(* PLC project Automatic_ScrewDriver_Line.project, CODESYS CODESYS V3.5 SP21 Patch 5 *)
(* stored: creationDateTime 2026-09-30T17:02:56.3790076, modificationDateTime 2026-09-30T17:02:44.4882995 *)

{attribute 'qualified_only'}
{attribute 'strict'}
TYPE JobState : (Idle := 1, Reset, ReadingTargetPosition, MovingToTargetPosition, MovingToBase, MovingZaxisToTool, ProcessingTool, MovingZaxisToBase, Error);
END_TYPE

TYPE Screw : STRUCT
  PositionMm : REAL;  (* in mm *)
  AngleDeg : DINT;  (* in ° *)
END_STRUCT;
END_TYPE

{attribute 'qualified_only'}
{attribute 'strict'}
TYPE ErrorCode : (NoError := 0, EnablementError, ScrewNotReleased, TargetNotReached, SpindleError, CobotNotConnected, CobotMovementNotReached, RtcNotAvailable);
END_TYPE

{attribute 'qualified_only'}
{attribute 'strict'}
TYPE ActionResult : (Busy := 1, Done, Failed);
END_TYPE

{attribute 'qualified_only'}
{attribute 'strict'}
TYPE MoverState : (Idle := 0, WaitingEcho, Moving, WaitingDoneReleased);
END_TYPE

TYPE JobReport : STRUCT
  JobId : UDINT;
  StartedAt : DT;
  FinishedAt : DT;
  ScrewsOk : INT;
  ScrewsFailed : INT;
  FailedScrews : ScrewList;
  Completed : BOOL;  (* TRUE = all screws processed, FALSE = aborted by operator *)
END_STRUCT;
END_TYPE

TYPE ScrewList : ARRAY[1..5] OF Screw;
END_TYPE

INTERFACE I_Actuator
METHOD Enable : BOOL
END_METHOD
METHOD Disable : BOOL
END_METHOD
END_INTERFACE

INTERFACE I_Mover
METHOD MoveToPosition : BOOL
  VAR_INPUT
    Position : REAL;
  END_VAR
END_METHOD
END_INTERFACE

INTERFACE I_Tool
METHOD ProcessTool : BOOL
  VAR_INPUT
    Angle : DINT;
  END_VAR
END_METHOD
END_INTERFACE

INTERFACE I_Resettable
METHOD Reset : BOOL
END_METHOD
END_INTERFACE

INTERFACE I_Diagnosable
METHOD GetError : ErrorCode
END_METHOD
METHOD ClearError : BOOL
END_METHOD
END_INTERFACE

INTERFACE I_ReportSink
METHOD PublishReport : BOOL
  VAR_INPUT
    Report : JobReport;
  END_VAR
END_METHOD
END_INTERFACE

INTERFACE I_Device
END_INTERFACE

PROGRAM PLC_PRG
  VAR
    _InitDone : BOOL;
    _JobManager : FB_JobManager;
    _UserInterface : FB_UserInterface;
    _JobSelector : FB_JobSelector;
    _Conveyor : FB_ConveyorElectrical;
    _Cobot : FB_Cobot;
    _zAxis : FB_zAxis;
    _Spindle : FB_Spindle;
    _ReportJob : FB_ReportJob;
    _LogSink : FB_LogSink;
  END_VAR

                    IF NOT _InitDone THEN
	_InitDone := InitPous();
END_IF


_JobManager.RunJob();


//I/O's connection: Machine -> Material
//For Conveyor:
IO_Simulation.MoverEnable := _Conveyor.MoverEnable;
IO_Simulation.MoverExecuteFor :=  _Conveyor.MoverExecuteFor;
IO_Simulation.MoverExecuteBac :=  _Conveyor.MoverExecuteBac;
// For Robot:
IO_Cobot.Cmd_TargetPos01mm := INT_TO_WORD(_Cobot.MoverTarget);   // 0..5000: no sign issue
IO_Cobot.Cmd_Start := _Cobot.MoverExecute;
IO_Cobot.Cmd_Enable := _Cobot.MoverEnable;
// For Z valve
IO_Simulation.zValve := _zAxis.zValve;
// For Spindle
IO_Simulation.SpindleEnable := _Spindle.SpindleEnable;
IO_Simulation.SpindleExecute := _Spindle.SpindleExecute;
IO_Simulation.SpindleExecuteTime := _Spindle.SpindleExecuteTime;

// Simulation
PRG_PlantSim();

//I/O's connection: Material -> Machine
//For Conveyor:
_Conveyor.MoverActPos := IO_Simulation.MoverActPos;
_Conveyor.MoverReady := IO_Simulation.MoverReady; 
// For cobot:
_Cobot.MoverPosEcho := WORD_TO_INT(IO_Cobot.Sts_TargetPosEcho01mm);
_Cobot.MoverDone := IO_Cobot.Sts_Done;
_Cobot.MoverHeartbeat := WORD_TO_INT(IO_Cobot.Sts_Heartbeat);
// For Z valve
_zAxis.ScrewEngaged := IO_Simulation.ScrewEngaged;
_zAxis.ScrewReleased := IO_Simulation.ScrewReleased;
_zAxis.zDown := IO_Simulation.zDown;
// For Spindle
_Spindle.SpindleReady := IO_Simulation.SpindleReady;
_Spindle.SpindleDone := IO_Simulation.SpindleDone;




                  

METHOD InitPous : BOOL
  VAR
    _Mover : I_Mover;
  END_VAR
                          // Injection of dependencies
IF Machine_Constants.USE_COBOT THEN
	_Mover := _Cobot;
ELSE
	_Mover := _Conveyor;
END_IF

_ReportJob.AddSink(_LogSink);

InitPous := _JobManager.Init(
	UserInterface := _UserInterface,
	JobSelector := _JobSelector,
	Mover:= _Mover,
	zAxis := _zAxis,
	Spindle := _Spindle,
	ReportJob := _ReportJob);
                        
END_METHOD
END_PROGRAM

FUNCTION_BLOCK FB_FunctionBlock_Base IMPLEMENTS I_Resettable, I_Diagnosable
  VAR
    _Error : ErrorCode;
  END_VAR

                    
                  

{attribute 'abstract'}
METHOD Reset : BOOL
                          
                        
END_METHOD

METHOD RaiseError : BOOL
  VAR_INPUT
    Error : ErrorCode;
  END_VAR
                          RaiseError := FALSE;

IF _Error = ErrorCode.NoError THEN
	_Error := Error;
	Trace(CmpLog.LogClass.LOG_ERROR, ErrorCodeToString(Error));
	RaiseError := TRUE;
END_IF

                        
END_METHOD

METHOD GetError : ErrorCode
                          GetError := _Error;
                        
END_METHOD

METHOD ClearError : BOOL
                          _Error := ErrorCode.NoError;
ClearError := TRUE;
                        
END_METHOD

METHOD HasError : BOOL
                          HasError := (_Error <> ErrorCode.NoError);
                        
END_METHOD
END_FUNCTION_BLOCK

FUNCTION_BLOCK FB_JobManager EXTENDS FB_FunctionBlock_Base
  VAR
    _InitDone : BOOL;
    _state : JobState;
    _ActiveError : ErrorCode;
    _Stop : BOOL;
    _Reseters : ARRAY[1..6] OF I_Resettable;
    _Diagnosable : ARRAY[1..6] OF I_Diagnosable;
    _i : DINT;
    _UserInterface : REFERENCE TO FB_UserInterface;
    _JobSelector : REFERENCE TO FB_JobSelector;
    _Mover : I_Mover;
    _zAxis : REFERENCE TO FB_zAxis;
    _Spindle : REFERENCE TO FB_Spindle;
    _ReportJob : REFERENCE TO FB_ReportJob;
    _SpindleOk : BOOL;
    _MoverOk : BOOL;
  END_VAR

                    
                  

METHOD Reset : BOOL
                          ClearError();
Reset := TRUE;

                        
END_METHOD

METHOD Init : BOOL
  VAR_INPUT
    UserInterface : REFERENCE TO FB_UserInterface;
    JobSelector : REFERENCE TO FB_JobSelector;
    Mover : I_Mover;
    zAxis : REFERENCE TO FB_zAxis;
    Spindle : REFERENCE TO FB_Spindle;
    ReportJob : REFERENCE TO FB_ReportJob;
  END_VAR
                          _UserInterface REF= UserInterface;
_JobSelector REF= JobSelector;
_Mover := Mover;
_zAxis REF= zAxis;
_Spindle REF= Spindle;
_ReportJob REF= ReportJob;

// Reseters
_Reseters[1] := _UserInterface;
_Reseters[2] := _JobSelector;
_Reseters[3] := _Mover;
_Reseters[4] := _zAxis;
_Reseters[5] := _Spindle;
_Reseters[6] := _ReportJob;

// Diagnosable
_Diagnosable[1] := _UserInterface;
_Diagnosable[2] := _JobSelector;
_Diagnosable[3] := _Mover;
_Diagnosable[4] := _zAxis;
_Diagnosable[5] := _Spindle;
_Diagnosable[6] := _ReportJob;

_InitDone := TRUE;
Init := TRUE;
                        
END_METHOD

METHOD DisableAll : BOOL
                          _SpindleOk := _Spindle.Disable();
_MoverOk   := _Mover.Disable();
DisableAll := _SpindleOk AND _MoverOk;
                        
END_METHOD

METHOD EnableAll : BOOL
                          _SpindleOk := _Spindle.Enable();
_MoverOk   := _Mover.Enable();
EnableAll  := _SpindleOk AND _MoverOk;

                        
END_METHOD

METHOD ResetAll : BOOL
                          ResetAll := TRUE;

FOR _i := 1 TO UPPER_BOUND(_Reseters, 1) DO
    IF NOT _Reseters[_i].Reset() THEN
        ResetAll := FALSE;
    END_IF
END_FOR
                        
END_METHOD

METHOD CheckErrors : ErrorCode
                          CheckErrors := ErrorCode.NoError;

FOR _i := 1 TO UPPER_BOUND(_Diagnosable, 1) DO
    IF _Diagnosable[_i].GetError() <> ErrorCode.NoError
       AND CheckErrors = ErrorCode.NoError THEN
        CheckErrors := _Diagnosable[_i].GetError();
    END_IF
END_FOR
                        
END_METHOD

METHOD RunJob : BOOL
                          IF NOT _InitDone THEN
	RETURN;
END_IF

_ActiveError := CheckErrors();
_Stop := _UserInterface.IsStopRequired();
		  
IF _ActiveError <> ErrorCode.NoError AND _state <> JobState.Reset THEN
    _state := JobState.Error;
END_IF

IF _state <> JobState.Reset AND _state <> JobState.Error THEN
    EnableAll();
ELSE
    DisableAll();
END_IF

CASE _state OF
	JobState.Reset :
		IF ResetAll() THEN
			_state := JobState.Idle;
		END_IF
	JobState.Idle:
		IF _Stop THEN
			_state := JobState.Reset;
		ELSIF _zAxis.Retract() THEN
        	IF _UserInterface.IsStartRequired() THEN
            _ReportJob.Reset();
			_ReportJob.JobStart();
            _state := JobState.ReadingTargetPosition;
        	END_IF
    	END_IF
	JobState.ReadingTargetPosition :
		IF _JobSelector.ReturnScrew() THEN
			_state:= JobState.MovingToTargetPosition;
		ELSE
			_state := JobState.MovingToBase;
		END_IF
	JobState.MovingToTargetPosition :
		IF _Mover.MoveToPosition(_JobSelector.CurrentScrew.PositionMm) THEN
			_state:= JobState.MovingZaxisToTool;
		END_IF
	JobState.MovingZaxisToTool :
		    CASE _zAxis.Engage() OF
        		ActionResult.Done:
            		_state := JobState.ProcessingTool;
				ActionResult.Failed:
            		_ReportJob.FailScrew(_JobSelector.CurrentScrew);
					_state := JobState.MovingZaxisToBase;
    		END_CASE
	JobState.ProcessingTool :
		IF _Spindle.ProcessTool(_JobSelector.CurrentScrew.AngleDeg) THEN		
			_ReportJob.SuccessScrew(_JobSelector.CurrentScrew);
			_state:= JobState.MovingZaxisToBase;
		END_IF
	JobState.MovingZaxisToBase :
		IF _zAxis.Retract() THEN
			_state:= JobState.ReadingTargetPosition;
		END_IF
	JobState.MovingToBase :
		IF _Mover.MoveToPosition(0)  THEN
			_state := JobState.Idle;
			_ReportJob.JobEnd();
		END_IF
	JobState.Error :
		IF _Stop THEN
			_state := JobState.Reset;
		END_IF
END_CASE

// Stop during a job = abort: publish the partial report, then reset every component.
// The next Start begins a fresh job from the first screw.
IF _Stop
   AND _state <> JobState.Idle
   AND _state <> JobState.Reset
   AND _state <> JobState.Error THEN
	_ReportJob.JobAborted();
	_state := JobState.Reset;
END_IF

                        
END_METHOD
END_FUNCTION_BLOCK

FUNCTION_BLOCK FB_UserInterface EXTENDS FB_FunctionBlock_Base
  VAR_INPUT
    StartRequest : BOOL;
    StopRequest : BOOL;
  END_VAR
  VAR
    _Start_Trig : R_TRIG;
    _Stop_Trig : R_TRIG;
  END_VAR

                    
                  

METHOD Reset : BOOL
                          ClearError();
Reset := TRUE;
                        
END_METHOD

METHOD IsStartRequired : BOOL
                          _Start_Trig(CLK := StartRequest);
IsStartRequired := _Start_Trig.Q;

                        
END_METHOD

METHOD IsStopRequired : BOOL
                          _Stop_Trig(CLK := StopRequest);
IsStopRequired := _Stop_Trig.Q;
                        
END_METHOD
END_FUNCTION_BLOCK

FUNCTION_BLOCK FB_JobSelector EXTENDS FB_FunctionBlock_Base
  VAR_INPUT
    ArrScrews : ScrewList := [(PositionMm := 100.0, AngleDeg := 90), (PositionMm := 130.0, AngleDeg := 600), (PositionMm := 185.0, AngleDeg := -180), (PositionMm := 27.0, AngleDeg := 360), (PositionMm := 300.0, AngleDeg := 720)];
  END_VAR
  VAR_OUTPUT
    CurrentScrew : Screw;
    Job_Done : BOOL;
  END_VAR
  VAR
    _TableIndex : INT := 0;
  END_VAR

                    
                  

METHOD Reset : BOOL
                          ClearError();
_TableIndex := 0;
Job_Done := FALSE;

Reset := TRUE;
                        
END_METHOD

METHOD ReturnScrew : BOOL
                          ReturnScrew := FALSE;


IF SelectNextScrew() THEN
	CurrentScrew := ArrScrews[_TableIndex];
	ReturnScrew := TRUE;
ELSE
	CurrentScrew.PositionMm := 0.0;
	CurrentScrew.AngleDeg := 0;
END_IF

                        
END_METHOD

METHOD SelectNextScrew : BOOL
                          // Method responsible for incrementing _TableIndex
SelectNextScrew := FALSE;
Job_Done := FALSE;
IF _TableIndex < UPPER_BOUND(ArrScrews, 1) THEN
	_TableIndex := _TableIndex + 1;
	SelectNextScrew := TRUE;
ELSE
	_TableIndex := 0;
	Job_Done := TRUE;
END_IF
                        
END_METHOD
END_FUNCTION_BLOCK

FUNCTION_BLOCK FB_ConveyorElectrical EXTENDS FB_FunctionBlock_Base IMPLEMENTS I_Mover
  VAR_INPUT
    MoverActPos : REAL;
    MoverReady : BOOL;
  END_VAR
  VAR_OUTPUT
    MoverEnable : BOOL;
    MoverExecuteFor : BOOL;
    MoverExecuteBac : BOOL;
  END_VAR
  VAR
    _MoverTarget : REAL;
    _TimerEnablement : TON;
    _TimerMoveLinear : TON;
  END_VAR

                    
                  

METHOD Reset : BOOL
                          ClearError();
Disable();
MoverExecuteFor := FALSE;
MoverExecuteBac := FALSE;
_MoverTarget :=  0.0;
_TimerEnablement(IN := FALSE, PT := T#1S);
_TimerMoveLinear(IN := FALSE, PT := T#100S);
Reset := TRUE;
                        
END_METHOD

METHOD MoveToPosition : BOOL
  VAR_INPUT
    Position : REAL;
  END_VAR
                          MoveToPosition := FALSE;

_MoverTarget := Position;


IF _TimerMoveLinear.Q THEN
	RaiseError(ErrorCode.TargetNotReached);
ELSIF _MoverTarget - MoverActPos >= 1 THEN
	MoverExecuteFor := TRUE;
ELSIF _MoverTarget - MoverActPos <= -1 THEN
	MoverExecuteBac := TRUE;
ELSE
	MoveToPosition := TRUE;
	MoverExecuteFor := FALSE;
	MoverExecuteBac := FALSE;
END_IF

_TimerMoveLinear(IN := (MoverExecuteFor OR MoverExecuteBac), PT := T#100S);

                        
END_METHOD

METHOD Enable : BOOL
                          Enable := FALSE;

MoverEnable := TRUE;
_TimerEnablement(IN := MoverEnable AND NOT MoverReady, PT := T#1S);

IF MoverReady THEN
	Enable := TRUE;
ELSIF _TimerEnablement.Q THEN
	RaiseError(ErrorCode.EnablementError);
END_IF

                        
END_METHOD

METHOD Disable : BOOL
                          MoverEnable := FALSE;
Disable := TRUE;
                        
END_METHOD
END_FUNCTION_BLOCK

FUNCTION_BLOCK FB_zAxis EXTENDS FB_FunctionBlock_Base
  VAR_INPUT
    zDown : BOOL;
    ScrewEngaged : BOOL;
    ScrewReleased : BOOL;
  END_VAR
  VAR_OUTPUT
    zValve : BOOL;
  END_VAR
  VAR
    _timerUp : TON;
    _timerDown : TON;
  END_VAR

                    
                  

METHOD Reset : BOOL
                          ClearError();

zValve := FALSE;

IF zDown THEN
	Reset := TRUE;
END_IF

_timerUp(IN := FALSE, PT := T#5S);
_timerDown(IN := FALSE, PT := T#5S);
                        
END_METHOD

METHOD Engage : ActionResult
                          Engage := ActionResult.Busy;
zValve := TRUE;

_timerUp(IN := zValve AND NOT ScrewEngaged, PT := T#5S);
_timerDown(IN := FALSE, PT := T#5S);

IF ScrewEngaged THEN
	Engage := ActionResult.Done;
ELSIF _timerUp.Q THEN
	Engage := ActionResult.Failed;
END_IF


                        
END_METHOD

METHOD Retract : BOOL
                          Retract := FALSE;
zValve := FALSE;

_timerDown(IN := NOT zValve AND NOT (zDown AND ScrewReleased), PT := T#5S);
_timerUp(IN := FALSE, PT := T#5S);

IF zDown AND ScrewReleased THEN
    Retract := TRUE;
ELSIF _timerDown.Q THEN
	RaiseError(ErrorCode.ScrewNotReleased);
END_IF


                        
END_METHOD
END_FUNCTION_BLOCK

FUNCTION_BLOCK FB_Spindle EXTENDS FB_FunctionBlock_Base IMPLEMENTS I_Actuator
  VAR_INPUT
    SpeedDegPerSec : DINT := Machine_Constants.TOOL_SPEED;
    SpindleReady : BOOL;
    SpindleDone : BOOL;
  END_VAR
  VAR_OUTPUT
    SpindleEnable : BOOL;
    SpindleExecute : BOOL;
    SpindleExecuteTime : TIME;
  END_VAR
  VAR
    _AngleTarget : DINT;
    _Started : BOOL;
    _TimerEnablement : TON;
    _TimerProcessTool : TON;
  END_VAR

                    
                  

METHOD Reset : BOOL
                          ClearError();
Disable();
SpindleEnable := FALSE;
SpindleExecute := FALSE;
SpindleExecuteTime := T#0S;
_AngleTarget := 0;
_Started := FALSE;
_TimerEnablement(IN := FALSE, PT := T#1S);
_TimerProcessTool(IN := FALSE, PT := T#20S);
Reset := TRUE;
                        
END_METHOD

METHOD ProcessTool : BOOL
  VAR_INPUT
    Angle : DINT;
  END_VAR
                          ProcessTool := FALSE;
_TimerProcessTool(IN := SpindleExecute AND NOT SpindleDone, PT := T#20S);
_AngleTarget := ABS(Angle); 

IF NOT _Started AND SpindleEnable THEN
	SpindleExecuteTime := DINT_TO_TIME(_AngleTarget*1000/SpeedDegPerSec);
	SpindleExecute := TRUE;
	_Started := TRUE;
ELSIF SpindleDone THEN
	SpindleExecute := FALSE;
	_Started := FALSE;
	ProcessTool := TRUE;
ELSIF _TimerProcessTool.Q THEN
	RaiseError(ErrorCode.SpindleError);
END_IF


                        
END_METHOD

METHOD Enable : BOOL
                          Enable := FALSE;

SpindleEnable := TRUE;
_TimerEnablement(IN := SpindleEnable AND NOT SpindleReady, PT := T#1S);

IF SpindleReady THEN
	Enable := TRUE;
ELSIF _TimerEnablement.Q THEN
	RaiseError(ErrorCode.EnablementError);
END_IF
                        
END_METHOD

METHOD Disable : BOOL
                          SpindleEnable := FALSE;
Disable := TRUE;
                        
END_METHOD
END_FUNCTION_BLOCK

PROGRAM PRG_PlantSim
  VAR
    _Increment : REAL := 1;
    _ZAxisMovingTimeUp : TON;
    _ZAxisMovingTimeDown : TON;
    _SpindleMovingTime : TON;
  END_VAR

                    // Conveyor
IO_Simulation.MoverReady := IO_Simulation.MoverEnable
                                   AND NOT IO_Simulation.SimFail_MoverReady;
IF IO_Simulation.MoverExecuteFor AND IO_Simulation.MoverEnable
   AND NOT IO_Simulation.SimFail_MoverBlocked THEN
    IO_Simulation.MoverActPos := IO_Simulation.MoverActPos + _Increment;
ELSIF IO_Simulation.MoverExecuteBac AND IO_Simulation.MoverEnable
   AND NOT IO_Simulation.SimFail_MoverBlocked THEN
    IO_Simulation.MoverActPos := IO_Simulation.MoverActPos - _Increment;
END_IF

// Z Axis
_ZAxisMovingTimeUp(IN := IO_Simulation.zValve, PT := T#1S);
IO_Simulation.ScrewEngaged := _ZAxisMovingTimeUp.Q
                                     AND NOT IO_Simulation.SimFail_ScrewEngaged;
_ZAxisMovingTimeDown(IN := NOT IO_Simulation.zValve, PT := T#1S);
IO_Simulation.ScrewReleased := _ZAxisMovingTimeDown.Q
                                      AND NOT IO_Simulation.SimFail_ScrewReleased;
// zDown is not filtered: the cylinder physically retracts even if the bit stays engaged
IO_Simulation.zDown := _ZAxisMovingTimeDown.Q;

// Spindle
IO_Simulation.SpindleReady := IO_Simulation.SpindleEnable;
_SpindleMovingTime(IN := IO_Simulation.SpindleExecute
                         AND IO_Simulation.SpindleEnable,
                   PT := IO_Simulation.SpindleExecuteTime);
IO_Simulation.SpindleDone := _SpindleMovingTime.Q
                                    AND NOT IO_Simulation.SimFail_SpindleDone;
                  
END_PROGRAM

FUNCTION_BLOCK FB_ReportJob EXTENDS FB_FunctionBlock_Base
  VAR
    _NbSuccess : INT := 0;
    _NbFail : INT := 0;
    _FailedScrews : ScrewList;
    _SuccessfulScrews : ScrewList;
    _JobDone : BOOL;
    _JobId : UDINT;
    _StartedAt : DT;
    _FinishedAt : DT;
    _Sinks : ARRAY[1..3] OF I_ReportSink;
    _EmptyScrewList : ScrewList;
  END_VAR

                    
                  

METHOD Reset : BOOL
                          ClearError();
_NbSuccess := 0;
_NbFail := 0;
_JobDone := FALSE;

_FailedScrews     := _EmptyScrewList;
_SuccessfulScrews := _EmptyScrewList;

Reset := TRUE;
                        
END_METHOD

METHOD JobEnd : BOOL
                          _FinishedAt := Now();

Trace(CmpLog.LogClass.LOG_INFO, 'Job Done');

JobEnd := SendReportToSinks(Completed := TRUE);
                        
END_METHOD

METHOD SuccessScrew : BOOL
  VAR_INPUT
    SuccessfulScrew : Screw;
  END_VAR
                          SuccessScrew := FALSE;

IF _NbSuccess < UPPER_BOUND(_SuccessfulScrews, 1) THEN
	_NbSuccess := _NbSuccess + 1;
	_SuccessfulScrews[_NbSuccess] := SuccessfulScrew;
	SuccessScrew := TRUE;
END_IF

Trace(CmpLog.LogClass.LOG_INFO,
        CONCAT('Screw successfully processed at position ', REAL_TO_STRING(SuccessfulScrew.PositionMm)));
                        
END_METHOD

METHOD FailScrew : BOOL
  VAR_INPUT
    FailedScrew : Screw;
  END_VAR
                          FailScrew := FALSE;

IF _NbFail < UPPER_BOUND(_FailedScrews, 1) THEN
	_NbFail := _NbFail + 1;
	_FailedScrews[_NbFail] := FailedScrew;
	FailScrew := TRUE;
END_IF

Trace(CmpLog.LogClass.LOG_WARNING,
        CONCAT('Screw missed at position ', REAL_TO_STRING(FailedScrew.PositionMm)));
                        
END_METHOD

METHOD JobStart : BOOL
                          _JobId      := _JobId + 1;
_StartedAt  := Now();
_FinishedAt := DT#1970-01-01-00:00:00;

Trace(CmpLog.LogClass.LOG_INFO, 'Job Started');

JobStart := TRUE;
                        
END_METHOD

METHOD JobAborted : BOOL
                          _FinishedAt := Now();

Trace(CmpLog.LogClass.LOG_WARNING, 'Job Aborted');

JobAborted := SendReportToSinks(Completed := FALSE);
                        
END_METHOD

METHOD AddSink : BOOL
  VAR_INPUT
    Sink : I_ReportSink;
  END_VAR
  VAR
    _i : DINT;
  END_VAR
                          AddSink := FALSE;

FOR _i := 1 TO UPPER_BOUND(_Sinks, 1) DO
	IF _Sinks[_i] = 0 THEN
		_Sinks[_i] := Sink;
		AddSink := TRUE;
		RETURN;
	END_IF
END_FOR
                        
END_METHOD

METHOD SendReportToSinks : BOOL
  VAR_INPUT
    Completed : BOOL;  (* TRUE = job finished normally, FALSE = aborted by operator *)
  END_VAR
  VAR
    _report : JobReport;
    _i : DINT;
  END_VAR
                          _report.JobId        := _JobId;
_report.StartedAt    := _StartedAt;
_report.FinishedAt   := _FinishedAt;
_report.ScrewsOk     := _NbSuccess;
_report.ScrewsFailed := _NbFail;
_report.FailedScrews := _FailedScrews;
_report.Completed := Completed;

SendReportToSinks := TRUE;

FOR _i := 1 TO UPPER_BOUND(_Sinks, 1) DO
	IF _Sinks[_i] <> 0 THEN
		IF NOT _Sinks[_i].PublishReport(_report) THEN
			SendReportToSinks := FALSE;
		END_IF
	END_IF
END_FOR
                        
END_METHOD

METHOD Now : DT
  VAR
    _sec : UDINT;
    _res : RTS_IEC_RESULT;
  END_VAR
                          _sec := SysTimeRtcGet(_res);

IF _res = Errors.ERR_OK THEN
	Now := UDINT_TO_DT(_sec);
ELSE
	Now := DT#1970-01-01-00:00:00;
	RaiseError(ErrorCode.RtcNotAvailable);
END_IF
                        
END_METHOD
END_FUNCTION_BLOCK

FUNCTION ErrorCodeToString : STRING
  VAR_INPUT
    Code : ErrorCode;
  END_VAR

                    CASE Code OF
	ErrorCode.NoError :
		ErrorCodeToString := 'No Error';
	ErrorCode.EnablementError:
		ErrorCodeToString := 'Enablement Error';
	ErrorCode.ScrewNotReleased:
		ErrorCodeToString := 'Screw Not Released';
	ErrorCode.TargetNotReached:
		ErrorCodeToString := 'Target Not Reached';
	ErrorCode.SpindleError:
		ErrorCodeToString := 'Spindle Error';
	ErrorCode.CobotNotConnected:
		ErrorCodeToString := 'Cobot Not Connected';
	ErrorCode.CobotMovementNotReached:
		ErrorCodeToString := 'Cobot Movement Not Reached';
	ErrorCode.RtcNotAvailable:
		ErrorCodeToString := 'Rtc Not Available';
ELSE
		ErrorCodeToString := 'Unknown Error';	
END_CASE
                  
END_FUNCTION

FUNCTION_BLOCK FB_Cobot EXTENDS FB_FunctionBlock_Base IMPLEMENTS I_Mover
  VAR_INPUT
    MoverPosEcho : INT;  (* Echo to ensure synchronisation with MoverTarget *)
    MoverDone : BOOL;
    MoverHeartbeat : INT;  (* Watchdog counter to make sure Cobot connection is not lost *)
  END_VAR
  VAR_OUTPUT
    MoverEnable : BOOL;
    MoverTarget : INT;
    MoverExecute : BOOL;
  END_VAR
  VAR
    _state : MoverState := MoverState.Idle;
    _TimerEcho : TON;
    _TimerMove : TON;
    _TimerEnablement : TON;
    _LastHeartbeat : INT;
    _HbTimer : TON;
    _Alive : BOOL;
    _HbChanged : BOOL;
  END_VAR

                    
                  

METHOD Reset : BOOL
                          ClearError();
Disable();
MoverTarget :=  0;
_state := MoverState.Idle;
_TimerEnablement(IN := FALSE, PT := T#1S);
_TimerEcho(IN := FALSE, PT := T#2S);
_TimerMove(IN := FALSE, PT := T#30S);
_HbTimer(IN := FALSE, PT := T#500MS);

Reset := TRUE;
                        
END_METHOD

METHOD MoveToPosition : BOOL
  VAR_INPUT
    Position : REAL;
  END_VAR
                          MoveToPosition := FALSE;

CASE _state OF

	MoverState.Idle:
		// Never start a cycle while the robot still asserts Done from a previous one
		IF NOT MoverDone THEN
			MoverTarget  := REAL_TO_INT(Position * 10.0);
			MoverExecute := FALSE;
			_state := MoverState.WaitingEcho;
		END_IF

	MoverState.WaitingEcho:
		IF MoverPosEcho = MoverTarget THEN
			MoverExecute := TRUE;
			_state := MoverState.Moving;
		ELSIF _TimerEcho.Q THEN
			RaiseError(ErrorCode.CobotNotConnected);
		END_IF

	MoverState.Moving:
		IF MoverDone THEN
			MoverExecute := FALSE;
			_state := MoverState.WaitingDoneReleased;
		ELSIF _TimerMove.Q THEN
			RaiseError(ErrorCode.CobotMovementNotReached);
		END_IF

	MoverState.WaitingDoneReleased:
		IF NOT MoverDone THEN
			MoveToPosition := TRUE;
			_state := MoverState.Idle;
		END_IF

END_CASE

_TimerEcho(IN := (_state = MoverState.WaitingEcho), PT := T#2S);
_TimerMove(IN := (_state = MoverState.Moving), PT := T#30S);

                        
END_METHOD

METHOD Enable : BOOL
                          _HbChanged := (MoverHeartbeat <> _LastHeartbeat);
_LastHeartbeat := MoverHeartbeat;
_HbTimer(IN := NOT _HbChanged, PT := T#500MS);
_Alive := NOT _HbTimer.Q;

Enable := FALSE;
MoverEnable := TRUE;

_TimerEnablement(IN := NOT _Alive, PT := T#1S);

IF _Alive THEN
	Enable := TRUE;
ELSIF _TimerEnablement.Q THEN
	RaiseError(ErrorCode.CobotNotConnected);
END_IF

                        
END_METHOD

METHOD Disable : BOOL
                          MoverEnable  := FALSE;
MoverExecute := FALSE;
Disable := TRUE;
                        
END_METHOD
END_FUNCTION_BLOCK

FUNCTION_BLOCK FB_LogSink IMPLEMENTS I_ReportSink

                    
                  

METHOD PublishReport : BOOL
  VAR_INPUT
    Report : JobReport;
  END_VAR
  VAR
    _msg : STRING(255);
  END_VAR
                          _msg := CONCAT('Job ', UDINT_TO_STRING(Report.JobId));
_msg := CONCAT(_msg,   ' finished: ');
_msg := CONCAT(_msg,   INT_TO_STRING(Report.ScrewsOk));
_msg := CONCAT(_msg,   ' ok, ');
_msg := CONCAT(_msg,   INT_TO_STRING(Report.ScrewsFailed));
_msg := CONCAT(_msg,   ' failed');

Trace(CmpLog.LogClass.LOG_INFO, _msg);

PublishReport := TRUE;
                        
END_METHOD
END_FUNCTION_BLOCK

FUNCTION Trace : BOOL
  VAR_INPUT
    Severity : UDINT;  (* LogClass.LOG_INFO / LOG_WARNING / LOG_ERROR *)
    Msg : STRING(255);
  END_VAR

                    LogAdd(
	hLogger   := CmpLog.LogConstants.LOG_STD_LOGGER,
	stCmpName := Machine_Constants.LOG_COMPONENT_NAME,
	diClassID := UDINT_TO_DINT(Severity),
	diErrorID := 0,
	diInfoID  := 0,
	stInfo    := Msg
);

Trace := TRUE;
                  
END_FUNCTION

CONFIGURATION Device
  RESOURCE Application ON PLC
    {attribute 'qualified_only'}
    VAR_GLOBAL  (* IO_Simulation *)
      MoverEnable : BOOL;  (* Mover Outputs: PLC to Machine *)
      MoverExecuteFor : BOOL;
      MoverExecuteBac : BOOL;
      MoverActPos : REAL;  (* Inputs: Machine to PLC *)
      MoverReady : BOOL;
      zValve : BOOL;  (* Z Axis Outputs: PLC to Machine *)
      zDown : BOOL;  (* Inputs: Machine to PLC *)
      ScrewEngaged : BOOL;
      ScrewReleased : BOOL;
      SpindleEnable : BOOL;  (* Spindle Outputs: PLC to Machine *)
      SpindleExecute : BOOL;
      SpindleExecuteTime : TIME;
      SpindleReady : BOOL;  (* Inputs: Machine to PLC *)
      SpindleDone : BOOL;
      SimFail_ScrewEngaged : BOOL;  (* Z axis rises but the bit never engages the screw *)
      SimFail_ScrewReleased : BOOL;  (* bit stays stuck in the screw head *)
      SimFail_SpindleDone : BOOL;  (* spindle never reports completion *)
      SimFail_MoverReady : BOOL;  (* drive never confirms torque *)
      SimFail_MoverBlocked : BOOL;  (* axis is commanded but does not move *)
    END_VAR
    {attribute 'qualified_only'}
    VAR_GLOBAL  (* IO_Cobot *)
      Cmd_Enable : BOOL;  (* Type Modbus: coil, Address: 18 *)
      Cmd_Start : BOOL;  (* Type Modbus: coil, Address: 16 *)
      Cmd_TargetPos01mm : WORD;  (* Type Modbus: register, Address: 128, unit 0.1mm (to keep .1mm resolution from Position) *)
      Sts_Done : BOOL;  (* Type Modbus: coil, Address: 17 *)
      Sts_TargetPosEcho01mm : WORD;  (* Type Modbus: register, Address: 129 *)
      Sts_Heartbeat : WORD;  (* Type Modbus: register, Address: 130 *)
    END_VAR
    {attribute 'qualified_only'}
    VAR_GLOBAL CONSTANT  (* Machine_Constants *)
      TOOL_SPEED : DINT := 60;  (* Speed of the spindle in deg/s *)
      USE_COBOT : BOOL := TRUE;  (* If FALSE then the conveyor is used instead *)
      LOG_COMPONENT_NAME : STRING := 'ScrewDriverLine';
    END_VAR
    TASK MainTask(INTERVAL := T#50ms, PRIORITY := 15);
    PROGRAM PLC_PRG WITH MainTask : PLC_PRG;
  END_RESOURCE
END_CONFIGURATION

CONFIGURATION Ethernet
END_CONFIGURATION

CONFIGURATION Modbus_TCP_Client_UniversalRobot
END_CONFIGURATION

CONFIGURATION Modbus_TCP_Server
END_CONFIGURATION
